(* IEC 61131-3 sources: CodesysTest/export/UN00 - Sharp Bagger/EM02 - Discharge/CM00 - Retracting Load Plate/FB_SimBasicLoadPlate.pou, 2 files *)

(* ---- FB_SimBasicLoadPlate.pou.st ---- *)
(*#-#-#-#-#-#-#-#-#-#---Declaration---#-#-#-#-#-#-#-#-#-#-#-#-#*)

FUNCTION_BLOCK FB_SimBasicLoadPlate EXTENDS FB_BaseComponent IMPLEMENTS IRetractingLoadPlate, IExecuteAutomatically
VAR_INPUT
	loadPlateDwell : REAL := 2.5;
END_VAR
VAR_OUTPUT
END_VAR
VAR
	beginDischarge : FB_SimulatedFeedback(name := CONCAT(_prefix,'Begin Discharge'));
END_VAR
(*#-#-#-#-#-#-#-#-#-#---Implementation---#-#-#-#-#-#-#-#-#-#-#-#-#*)

(* ---- ClearStatus.m.st ---- *)
(*#-#-#-#-#-#-#-#-#-#---Declaration---#-#-#-#-#-#-#-#-#-#-#-#-#*)

METHOD PRIVATE ClearStatus
VAR_INPUT
END_VAR
(*#-#-#-#-#-#-#-#-#-#---Implementation---#-#-#-#-#-#-#-#-#-#-#-#-#*)

beginDischarge.in := FALSE;
THIS^.Execute();
